TYPE ST_LaudaWriteCommands_Status :
STRUCT
	StartStop	: STRING := 'STARTSTOP';
END_STRUCT
END_TYPE

(* stored: Version 1.1.0.1, ProductVersion 3.1.4024.12
   DUT ST_LaudaWriteCommands_Status: Id {5d0b82e9-fdd1-48e1-b22b-6fd76299a00a} *)
